// TwinCAT 3 PLC project TCP_Server
// ProgramVersion: 3.1.4020.10
// libraries:
//   Tc2_Standard, * (Beckhoff Automation GmbH)
//   Tc2_System, * (Beckhoff Automation GmbH)
//   Tc2_TcpIp, * (Beckhoff Automation GmbH)
//   Tc3_Module, * (Beckhoff Automation GmbH)
// project tree:
//   DUTs/ E_State.TcDUT
//   / PlcTask.TcTTO (not stored)
//   POUs/ FB_TcpServer.TcPOU, MAIN.TcPOU, FB_Toggle.TcPOU
// real-time tasks:
//   TASK PlcTask: cycle T#10ms, priority 20, ADS port 350

// ---- DUTs/E_State.TcDUT
{attribute 'qualified_only'}
{attribute 'strict'}
TYPE E_State :
(
 	STATE_INIT,
	STATE_CONNECTING,
	STATE_RECEIVING_DATA,
	STATE_SENDING_DATA,
	STATE_PROCESSING_DATA,
	STATE_ERROR_CLOSE_LISTEN
);
END_TYPE

// ---- POUs/FB_TcpServer.TcPOU
FUNCTION_BLOCK FB_TcpServer
VAR_INPUT
	NetId				: STRING; 	(* address of the TwinCAT TCP/IP Connection Server. For the local computer (default) an empty string may be specified*)
	ServerAdr 			: STRING;	(* Local server IP address (Ipv4) as a string*)
	ServerPort 			: UDINT;	(* Local server IP port *)
	sSend 				: STRING;	(* String to be sent *)
END_VAR
VAR_OUTPUT
	sReceive			: STRING;	(* String received *)
	bBusy				: BOOL;
	err					: BOOL;
	errid				: UDINT;
END_VAR
VAR
	fbSocketCloseAll	: FB_SocketCloseAll :=  ( sSrvNetID := '', tTimeout := DEFAULT_ADS_TIMEOUT );
	bCloseAll			: BOOL := TRUE;
		
	Timeout 			: TIME := T#10S;
	fbSocketListen		: FB_SocketListen := (bExecute := TRUE);
	fbSocketReceive		: FB_SocketReceive;
	fbSocketAccept		: FB_SocketAccept;
	fbSocketSend 		: FB_SocketSend;
	hListen				: T_HSOCKET;
	hSocket				: T_HSOCKET;
    
	bConnAccepted		: BOOL;            	
	RxBuffer			: STRING;
	state				: E_State;
           	
	Pulse_timer				: TON;
END_VAR

IF bCloseAll THEN (*On PLC reset or program download close all old connections *)
	bCloseAll := FALSE;
	fbSocketCloseAll( bExecute:= TRUE );
ELSE
	fbSocketCloseAll( bExecute:= FALSE );
END_IF

IF sSend = '' THEN
	sSend := 'Default response';
END_IF
				
Pulse_timer(IN:= , PT:= T#100MS, Q=> , ET=> );

fbSocketListen(							// Open Listener-Socket
		sSrvNetId:= NetId, 			
		sLocalHost:= ServerAdr, 
		nLocalPort:= ServerPort, 
		bExecute:= , 					//The block is activated by a rising edge at this input.
		tTimeout:= Timeout, 			//Maximum time allowed for the execution of the function block
		bBusy=> bBusy, 					//When the function block is activated this output is set. It remains set until and acknowledgement is received
		bError=> err, 					// IF an error should occur during the transfer OF the command, THEN THIS output is set once the bBusy output was reset
		nErrId=> errid, 				// If the bError output is set ,this parameter returns error number
		hListener=> hListen);			// Connection handle for the new listener socket

fbSocketAccept(
		sSrvNetId:= NetId, 
		hListener:= hListen, 
		bExecute:= , 
		tTimeout:= Timeout, 
		bAccepted=> bConnAccepted, 		//This output is set if a new connection to a remote client was established
		bBusy=> bBusy, 
		bError=> err, 
		nErrId=> errid, 
		hSocket=> hSocket);				//Connection handle of a new remote client
	
fbSocketSend(
		sSrvNetId:= NetId, 
		hSocket:= hSocket, 				//connection handle of the communication partner to which data are to be sent.
		cbLen:= LEN(sSend), 			//number of data to be sent in bytes.
		pSrc:= ADR(sSend), 				//address (pointer) of the transmit buffer.
		bExecute:= , 
		tTimeout:= Timeout, 
		bBusy=> bBusy, 
		bError=> err, 
		nErrId=> errid);

fbSocketReceive(
		sSrvNetId:= NetId, 
		hSocket:= hSocket,				// Connection handle of the communication partner from which data are to be received. 
		cbLen:= SIZEOF(RxBuffer), 		//Maximum available buffer size in bytes for the data to be read.
		pDest:= ADR(RxBuffer), 			//Address (pointer) of the receive buffer.
		bExecute:= , 
		tTimeout:= Timeout, 
		bBusy=> bBusy, 
		bError=> err, 
		nErrId=> errid, 
		nRecBytes=> );					// Number of the last successfully receive data bytes
		
CASE state OF
	E_State.STATE_INIT:
		//Open the port
		fbSocketListen.bExecute := TRUE;
		state := E_State.STATE_CONNECTING;
		
		
	E_State.STATE_CONNECTING:
		fbSocketListen.bExecute := FALSE;
		//Accept incoming connection every half a second
		IF NOT fbSocketListen.bBusy AND NOT fbSocketListen.bError THEN
			fbSocketAccept.bExecute := FALSE;
			Pulse_timer.IN := TRUE;
	
			IF bConnAccepted THEN
				fbSocketReceive.bExecute := TRUE;
				state := E_State.STATE_RECEIVING_DATA;
			ELSIF Pulse_timer.Q THEN
				fbSocketAccept.bExecute := TRUE;
				Pulse_timer.IN := FALSE;
			END_IF
		END_IF
	
		
	E_State.STATE_RECEIVING_DATA:
		fbSocketReceive.bExecute := FALSE;
		
		IF NOT fbSocketReceive.bBusy AND NOT fbSocketReceive.bError THEN
			IF fbSocketReceive.nRecBytes = 0 THEN
				//if there's no data received, reset the fbSocketReceive
				fbSocketReceive.bExecute := TRUE;
			ELSE
				MEMSET(ADR(sReceive),0,SIZEOF(sReceive));
				MEMCPY(ADR(sReceive), fbSocketReceive.pDest, fbSocketReceive.nRecBytes);
				

				fbSocketSend.bExecute := TRUE;
				state := E_State.STATE_SENDING_DATA;
			END_IF
		END_IF
	
		
	E_State.STATE_SENDING_DATA:
		fbSocketSend.bExecute := FALSE;
		
		IF NOT fbSocketSend.bBusy AND NOT fbSocketSend.bError THEN 
				fbSocketReceive.bExecute := TRUE;
				state := E_State.STATE_RECEIVING_DATA;
		END_IF
END_CASE

END_FUNCTION_BLOCK

// ---- POUs/MAIN.TcPOU
PROGRAM MAIN
VAR
	fbTcpServer 	: FB_TcpServer;
	SrvNetId		: STRING := '';
	ServerAddress 	: STRING := '127.0.0.1';
	ServerPort 		: UDINT := 2000;
	
	sResponse		: STRING;
	sCommand		: STRING;
	bBusy			: BOOL;
	err				: BOOL;
	errid			: UDINT;
	
	Toggle 	: FB_Toggle;
	MemBit0 AT %MX0.0 : BOOL    := FALSE;
	
END_VAR

fbTcpServer(
	NetId:= SrvNetId, 
	ServerAdr:= ServerAddress, 
	ServerPort:= ServerPort, 
	sSend := sResponse,
	sReceive=> sCommand, 
	bBusy=> bBusy, 
	err=> err, 
	errid=> errid);

Toggle(Timer:= T#500MS , Toggle_Out=> );
MemBit0 := Toggle.Toggle_Out;

sResponse := sCommand;
IF sCommand = 'BIT-0' THEN
	IF MemBit0 THEN
		sResponse := '1';
	ELSE
		sResponse := '0';
	END_IF
END_IF

END_PROGRAM

// ---- POUs/FB_Toggle.TcPOU
FUNCTION_BLOCK FB_Toggle
VAR_INPUT
	Timer : TIME;
END_VAR
VAR_OUTPUT
	Toggle_Out : BOOL;
END_VAR
VAR
	Timer_Out : BOOL;
	Timer_Toggle: TON;
END_VAR

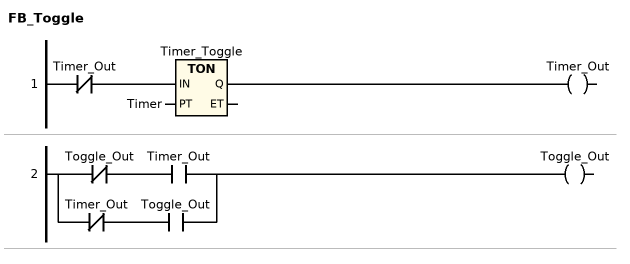
// NETWORK 1
Timer_Toggle(IN := NOT Timer_Out, PT := Timer); // TON
Timer_Out := Timer_Toggle.Q;

// NETWORK 2
Toggle_Out := NOT Toggle_Out AND Timer_Out OR NOT Timer_Out AND Toggle_Out;

END_FUNCTION_BLOCK
